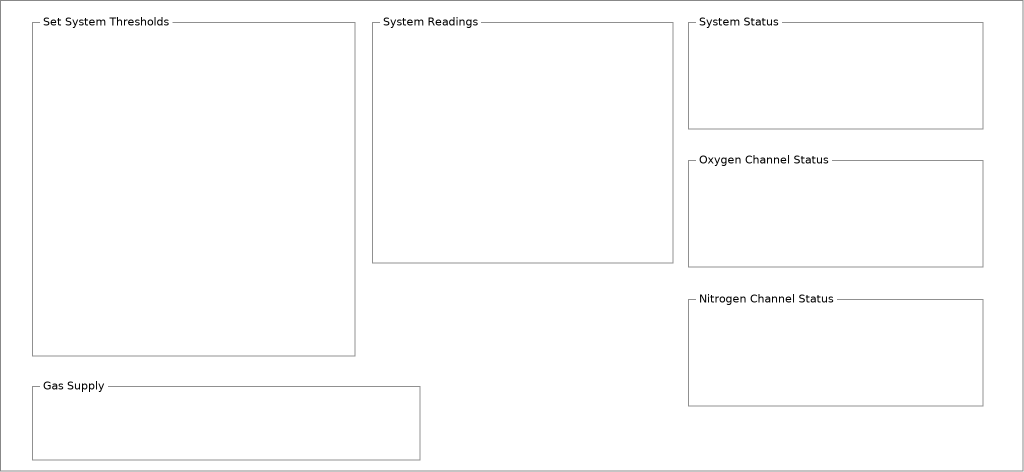
VISUALIZATION _003_Settings  // 1024x472
    GroupBox (32,378 388x82), "Gas Supply"
    GroupBox (32,14 323x342), "Set System Thresholds"
    GroupBox (372,14 301x249), "System Readings"
    GroupBox (688,14 295x115), "System Status"
    GroupBox (688,152 295x115), "Oxygen Channel Status"
    GroupBox (688,291 295x115), "Nitrogen Channel Status"
END_VISUALIZATION

(* stored: Version 1.1.0.1, ProductVersion 3.1.4022.18
   Visu _003_Settings: Id {f9370dbe-13d8-4f61-8a42-43d6707536f2} *)
